TYPE ST_PowerMonitor_OutputField EXTENDS st_MeasurementVoltageData:
STRUCT
	r_loadshare					: 	REAL;
	Powerlock					: 	ARRAY [1..3] OF ST_MeasurementFieldData;
END_STRUCT
END_TYPE

(* stored: Version 1.1.0.1, ProductVersion 3.1.4024.12
   DUT ST_PowerMonitor_OutputField: Id {d081661a-6cb9-4458-b0a8-f5a8c188d6d3} *)
